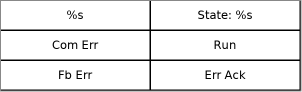
VISUALIZATION TplTsGroup  // 302x92
VAR_IN_OUT
	stGroupDiag					:FB_TwinSafeGroup;
END_VAR
(* End *)
    Rectangle (0,30 150x30), "Com Err", colour toggle: stGroupDiag.bComErr
    Rectangle (0,60 150x30), "Fb Err", colour toggle: stGroupDiag.bFbErr
    Rectangle (150,0 150x30), "State: %s", text variable: stGroupDiag.sState, colour toggle: stGroupDiag.sState = 'ERROR'
    Rectangle (150,30 150x30), "Run", colour toggle: stGroupDiag.bRun
    Rectangle (150,60 150x30), "Err Ack", colour toggle: stGroupDiag.bErrAck
    Rectangle (0,0 150x30), "%s", text variable: stGroupDiag.sName, colour toggle: stGroupDiag.sState = 'RUN'
END_VISUALIZATION

(* stored: Version 1.1.0.1
   Visu TplTsGroup: Id {e6422997-abbd-4b8c-b680-7a22b71b6303} *)
